# B&R Automation Studio project MotionTestBenchMaster (part 41)

```iecst
(* Input Signals *)
xInputAuto					:= stFillerModule.iq_stCmd.i_xAutoMode;
xInputJogMulti				:= stFillerModule.iq_stCmd.i_xJogMultiMode;
xInputAutoMulti				:= stFillerModule.iq_stCmd.i_xAutoMultiMode;
xInputSelHoming				:= stFillerModule.iq_stCmd.i_xSelectiveHomingMode;
xInputVelocity				:= stFillerModule.iq_stCmd.i_xVelocityMode;
xInputPositioning			:= stFillerModule.iq_stCmd.i_xPositioningMode;
xInputThirdPartySetup		:= stFillerModule.iq_stCmd.i_xThirdPartySetup;
xInputInductionSetup		:= stFillerModule.iq_stCmd.i_xInductionSetup;
xInputSlowMotion			:= stFillerModule.iq_stCmd.i_xSlowMotionForward OR stFillerModule.iq_stCmd.i_xSlowMotionBackward;
xInputBrakeRelease			:= stFillerModule.iq_stCmd.i_xBrakeRelease;
xInputStepByStep			:= stFillerModule.iq_stCmd.i_xStepByStep;
xInputStepByStepSingleAxis	:= stFillerModule.iq_stCmd.i_xStepByStepSingleAxis;//V4.A.A.1.7.0 Footbar
END_STEP
STEP ModeSelection:
(* Operating modes bits *)
xNoOpActive				:= TRUE;
xAutoActive 			:= FALSE;
xPositioningActive 		:= FALSE;
xSelHomingActive 		:= FALSE;
xBrakeReleaseActive 	:= FALSE;
xSlowMotionActive 		:= FALSE;
xJogMultiActive 		:= FALSE;
xAutoMultiActive 		:= FALSE;
xStepByStepActive 		:= FALSE;
xThirdPartySetupActive	:= FALSE;
xInductionSetupActive	:= FALSE;

(* Change status *)
xModeReady	:= usiMasterRequest = usiMasterStatus	AND
				NOT xAutoMode 						AND
				NOT xPositioningMode 				AND
				NOT xSelectiveHomingMode			AND
				NOT xVelocityMode					AND
				NOT xPositioningMode				AND
				NOT xStepByStepMode					AND
				NOT xJogMultiMode					AND
				NOT xAutoMultiMode					AND
				NOT xSlowMotionMode					AND
				NOT xThirdPartySetupMode			AND
				NOT xInductionSetupMode				AND
				NOT tofReactionActive.Q;

IF xModeReady THEN
	(* Local Master Request *)
	IF xInputJogMulti OR xInputAutoMulti THEN
		usiMasterRequest	:= LOCAL_MASTER;
	ELSIF xInputAuto OR	xInputPositioning OR xInputSelHoming OR xInputStepByStep OR xInputVelocity OR xInputThirdPartySetup OR xInputInductionSetup THEN
		usiMasterRequest	:= GLOBAL_MASTER;
	END_IF

	IF usiMasterStatus = GLOBAL_MASTER THEN
		IF xInputAuto THEN
			xAutoMode				:= TRUE;
		ELSIF xInputPositioning THEN
			xPositioningMode		:= TRUE;
		ELSIF xInputSelHoming THEN
			xSelectiveHomingMode	:= TRUE;
		ELSIF xInputThirdPartySetup THEN
			xThirdPartySetupMode	:= TRUE;
		ELSIF xInputInductionSetup THEN
			xInductionSetupMode		:= TRUE;
		ELSIF xInputStepByStep THEN
			xStepByStepMode			:= TRUE;
		ELSIF xInputVelocity THEN
			xVelocityMode			:= TRUE;
		END_IF
	ELSIF usiMasterStatus = LOCAL_MASTER THEN
		IF xInputJogMulti THEN
			xJogMultiMode 			:= TRUE;
		ELSIF xInputAutoMulti THEN
			xAutoMultiMode 			:= TRUE;
		ELSIF xInputSlowMotion THEN
			xSlowMotionMode			:= TRUE;
		END_IF
	END_IF
ELSIF tofReactionActive.Q THEN
	xBrakeReleaseMode	:= xInputBrakeRelease;
END_IF
END_STEP
ENTRY_ACTION
xExitStep	:= FALSE;
uiAutoStep	:= 0;
stFillerModule.iq_stStatus.q_xMasterRephased := FALSE;
END_ACTION
EXIT_ACTION
xNoOpActive	:= FALSE;
END_ACTION
TRANSITION FROM ModeSelection TO Auto:=
xAutoMode
END_TRANSITION
TRANSITION FROM ModeSelection TO Positioning:=
xPositioningMode
END_TRANSITION
STEP Positioning:
IF xReactionActive OR NOT xInputPositioning THEN
	xPositioningMode	:= FALSE;
END_IF

xPositioningActive	:= TRUE;

CASE uiPositioningStep OF
	0:
		IF stFillerModule.iq_stStatus.q_xRealAxesReadyForACommand AND stFillerModule.iq_astSubModuleAxis[CST_ModuleMasterAxis].iq_stStatus.q_stMainAxisStatus.q_xReadyForACommand THEN
			IF NOT stFillerModule.iq_stStatus.q_xSynchroWithOffset THEN
				uiPositioningStep	:= 100;
			ELSE
				uiPositioningStep	:= 50;
			END_IF
		END_IF

	50:
		FOR uiAxisIndex	:= uiFirstFillerModuleAxis TO uiLastFillerModuleAxis BY 1 DO
			stFillerModule.iq_astSubModuleAxis[uiAxisIndex].iq_stCmd.i_xPhaseCompensation := stFillerModule.iq_astSubModuleAxis[uiAxisIndex].iq_stStatus.q_stMainAxisStatus.q_xSynchroWithOffset;
		END_FOR

		IF NOT stFillerModule.iq_stStatus.q_xSynchroWithOffset THEN
			uiPositioningStep := 60;
		END_IF

	60:
		FOR uiAxisIndex	:= uiFirstFillerModuleAxis TO uiLastFillerModuleAxis BY 1 DO
			stFillerModule.iq_astSubModuleAxis[uiAxisIndex].iq_stCmd.i_xPhaseCompensation := FALSE;
		END_FOR
		uiPositioningStep := 100;

	100:
		IF stFillerModule.iq_stParameters.i_uiAxisSelected >= uiFirstFillerModuleAxis AND stFillerModule.iq_stParameters.i_uiAxisSelected <= uiLastFillerModuleAxis THEN
			uiOldAxisSelected := stFillerModule.iq_stParameters.i_uiAxisSelected;
			IF stFillerModule.iq_astSubModuleAxis[uiOldAxisSelected].iq_stStatus.q_stMainAxisStatus.q_xAxisReal THEN
				uiPositioningStep := 110;
			END_IF
		END_IF

	110:
		IF stFillerModule.iq_stCmd.i_xStepByStepSingleAxis THEN //V4.A.A.1.7.0 Footbar
			stFillerModule.iq_astSubModuleAxis[uiOldAxisSelected].iq_stParam.i_rPositioningVelocity	:= 10 * CST_PositioningVel ;
			stFillerModule.iq_astSubModuleAxis[uiOldAxisSelected].iq_stParam.i_rPositioningAccDec	:= 3 * CST_PositioningAccDec;
			stFillerModule.iq_astSubModuleAxis[uiOldAxisSelected].iq_stParam.i_lrAdditiveDistance	:= stFillerModule.iq_stParameters.i_rPositioningOffset;
		ELSE
			stFillerModule.iq_astSubModuleAxis[uiOldAxisSelected].iq_stParam.i_rPositioningVelocity	:= CST_PositioningVel;
			stFillerModule.iq_astSubModuleAxis[uiOldAxisSelected].iq_stParam.i_rPositioningAccDec	:= CST_PositioningAccDec;
			stFillerModule.iq_astSubModuleAxis[uiOldAxisSelected].iq_stParam.i_lrAdditiveDistance	:= stFillerModule.iq_stParameters.i_rPositioningOffset;
		END_IF

		IF stFillerModule.iq_astSubModuleAxis[uiOldAxisSelected].iq_stParam.i_lrAdditiveDistance = 0 THEN
			stFillerModule.iq_astSubModuleAxis[uiOldAxisSelected].iq_stParam.i_lrAdditiveDistance := 360.0;
		END_IF

		stFillerModule.iq_astSubModuleAxis[uiOldAxisSelected].iq_stCmd.i_xMoveAdditive	:= TRUE;

		tonPositDone(IN := FALSE, PT := T#5s);
		uiPositioningStep := 120;

	120:
		tonPositDone(IN := TRUE, PT := T#5s);
		IF NOT stFillerModule.iq_stStatus.q_xModuleStopped OR tonPositDone.Q THEN
			uiPositioningStep := 130;
		END_IF

	130:
		IF stFillerModule.iq_stStatus.q_xModuleStopped THEN
			stFillerModule.iq_astSubModuleAxis[uiOldAxisSelected].iq_stCmd.i_xMoveAdditive := FALSE;
			uiPositioningStep := 140;
		END_IF

	140:
		stFillerModule.iq_stStatus.q_xPositioningDone := TRUE;
END_CASE
END_STEP
ENTRY_ACTION
uiPositioningStep	:= 0;
END_ACTION
EXIT_ACTION
stFillerModule.iq_stStatus.q_xPositioningDone := FALSE;
stFillerModule.iq_astSubModuleAxis[uiOldAxisSelected].iq_stParam.i_rPositioningVelocity	:= CST_PositioningVel;//V4.A.A.1.7.0 Footbar
stFillerModule.iq_astSubModuleAxis[uiOldAxisSelected].iq_stParam.i_rPositioningAccDec	:= CST_PositioningAccDec;//V4.A.A.1.7.0 Footbar
END_ACTION
TRANSITION FROM Positioning TO PositExit:=
NOT xPositioningMode
END_TRANSITION
STEP PositExit:
stFillerModule.iq_astSubModuleAxis[uiOldAxisSelected].iq_stCmd.i_xMoveAdditive := FALSE;
stFillerModule.iq_stStatus.q_xPositioningDone := FALSE;
xExitStep := TRUE;
END_STEP
TRANSITION FROM PositExit TO ModeSelection:=
xExitStep
END_TRANSITION
(* @SFCISJUMP := 'ModeSelection' *)
TRANSITION FROM ModeSelection TO Velocity:=
xVelocityMode
END_TRANSITION
STEP Velocity:
IF xReactionActive OR NOT xInputVelocity THEN
	xVelocityMode	:= FALSE;
END_IF

xVelocityActive	:= TRUE;

CASE uiVelocityStep OF
	0:
		IF stFillerModule.iq_stStatus.q_xRealAxesReadyForACommand THEN
			uiVelocityStep	:= 100;
		END_IF

	100:
		IF stFillerModule.iq_stParameters.i_uiAxisSelected >= uiFirstFillerModuleAxis AND stFillerModule.iq_stParameters.i_uiAxisSelected <= uiLastFillerModuleAxis THEN
			uiOldAxisSelected	:= stFillerModule.iq_stParameters.i_uiAxisSelected;
			IF stFillerModule.iq_astSubModuleAxis[uiOldAxisSelected].iq_stStatus.q_stMainAxisStatus.q_xAxisReal THEN
				uiVelocityStep	:= 110;
			END_IF
		END_IF

	110:
		stFillerModule.iq_astSubModuleAxis[uiOldAxisSelected].iq_stParam.i_rEndlessVelocity		:= stFillerModule.iq_stParameters.i_rManualVelocity;

		stFillerModule.iq_astSubModuleAxis[uiOldAxisSelected].iq_stParam.i_lrAdditiveDistance	:= stFillerModule.iq_stParameters.i_rPositioningOffset;
		stFillerModule.iq_astSubModuleAxis[uiOldAxisSelected].iq_stCmd.i_xMoveVelocity			:= stFillerModule.iq_stCmd.i_xStart;
		uiVelocityStep	:= 120;

	120:
END_CASE
END_STEP
ENTRY_ACTION
uiVelocityStep	:= 0;
END_ACTION
EXIT_ACTION
xVelocityActive		:= FALSE;
uiOldAxisSelected	:= LIMIT(CST_FirstFillerModuleAxis, uiOldAxisSelected, CST_LastFillerModuleAxis);
stFillerModule.iq_astSubModuleAxis[uiOldAxisSelected].iq_stCmd.i_xMoveVelocity	:= FALSE;
END_ACTION
TRANSITION FROM Velocity TO VelExit:=
NOT xVelocityMode
END_TRANSITION
STEP VelExit:
xExitStep	:= stFillerModule.iq_stStatus.q_xModuleStopped;
END_STEP
TRANSITION FROM VelExit TO ModeSelection:=
xExitStep
END_TRANSITION
(* @SFCISJUMP := 'ModeSelection' *)
TRANSITION FROM ModeSelection TO SelHome:=
xSelectiveHomingMode
END_TRANSITION
STEP SelHome:
IF xReactionActive OR NOT xInputSelHoming THEN
	xSelectiveHomingMode := FALSE;
END_IF

xSelHomingActive	:= TRUE;

CASE uiSelectiveHomeStep OF
	0:
		IF stFillerModule.iq_stParameters.i_uiAxisSelected >= uiFirstFillerModuleAxis AND stFillerModule.iq_stParameters.i_uiAxisSelected <= uiLastFillerModuleAxis THEN
			uiOldAxisSelected	:= stFillerModule.iq_stParameters.i_uiAxisSelected;
			IF stFillerModule.iq_astSubModuleAxis[uiOldAxisSelected].iq_stStatus.q_stMainAxisStatus.q_xAxisReal THEN
				uiSelectiveHomeStep	:= 10;
			END_IF
		END_IF

	10:
		stFillerModule.iq_astSubModuleAxis[uiOldAxisSelected].iq_stCmd.i_xHome	:= TRUE;
		IF NOT stFillerModule.iq_astSubModuleAxis[uiOldAxisSelected].iq_stStatus.q_stMainAxisStatus.q_xIsHomed THEN
			uiSelectiveHomeStep	:= 20;
		END_IF

	20:
		uiSelectiveHomeStep	:= 30;

	30:
		IF stFillerModule.iq_astSubModuleAxis[uiOldAxisSelected].iq_stStatus.q_stMainAxisStatus.q_xIsHomed THEN
			stFillerModule.iq_astSubModuleAxis[uiOldAxisSelected].iq_stCmd.i_xHome	:= FALSE;
			uiSelectiveHomeStep	:= 40;
		END_IF

	40:
		stFillerModule.iq_stStatus.q_xSelHomingDone	:= TRUE;
END_CASE
END_STEP
ENTRY_ACTION
uiSelectiveHomeStep	:= 0;

(* Selective Homing done *)
stFillerModule.iq_stStatus.q_xSelHomingDone	:= FALSE;
END_ACTION
EXIT_ACTION
(* Selective Homing done *)
stFillerModule.iq_stStatus.q_xSelHomingDone	:= FALSE;
END_ACTION
TRANSITION FROM SelHome TO SelHomeExit:=
NOT xSelectiveHomingMode
END_TRANSITION
STEP SelHomeExit:
stFillerModule.iq_astSubModuleAxis[uiOldAxisSelected].iq_stCmd.i_xHome	:= FALSE;
xExitStep	:= TRUE;
END_STEP
TRANSITION FROM SelHomeExit TO ModeSelection:=
xExitStep
END_TRANSITION
(* @SFCISJUMP := 'ModeSelection' *)
TRANSITION FROM ModeSelection TO Brake:=
xBrakeReleaseMode
END_TRANSITION
STEP Brake:
xBrakeReleaseActive	:= TRUE;

IF NOT xInputBrakeRelease THEN
	xBrakeReleaseMode	:= FALSE;
END_IF

xBrakeReleaseActive	:= TRUE;

CASE uiBrakeReleaseStep OF
	0:
		uiOldAxisSelected	:= 0;
		IF stFillerModule.iq_stParameters.i_uiAxisSelected >= uiFirstFillerModuleAxis AND stFillerModule.iq_stParameters.i_uiAxisSelected <= uiLastFillerModuleAxis THEN
			uiOldAxisSelected	:= stFillerModule.iq_stParameters.i_uiAxisSelected;
			IF stFillerModule.iq_astSubModuleAxis[uiOldAxisSelected].iq_stStatus.q_stMainAxisStatus.q_xAxisReal THEN
				IF stFillerModule.iq_astSubModuleAxis[uiOldAxisSelected].iq_stStatus.q_stMainAxisStatus.q_xMotorWithBrake THEN
					uiBrakeReleaseStep	:= 100;
				ELSE
					uiBrakeReleaseStep	:= 400;
				END_IF
			END_IF
		END_IF

	100:
		stFillerModule.iq_astSubModuleAxis[uiOldAxisSelected].iq_stCmd.i_xReleaseBrake	:= TRUE;
		IF stFillerModule.iq_astSubModuleAxis[uiOldAxisSelected].iq_stStatus.q_stMainAxisStatus.q_xBrakeReleased THEN
			uiBrakeReleaseStep	:= 200;
		END_IF

	200:
		stFillerModule.iq_stStatus.q_xBrakeReleaseDone	:= TRUE;

	400:
		stFillerModule.iq_stStatus.q_xBrakeReleaseDone	:=	TRUE;
END_CASE
END_STEP
ENTRY_ACTION
uiBrakeReleaseStep	:= 0;
END_ACTION
EXIT_ACTION
xBrakeReleaseActive	:= FALSE;
stFillerModule.iq_stStatus.q_xBrakeReleaseDone	:= FALSE;

IF uiOldAxisSelected <> 0 THEN
	stFillerModule.iq_astSubModuleAxis[uiOldAxisSelected].iq_stCmd.i_xReleaseBrake	:= FALSE;
END_IF
END_ACTION
TRANSITION FROM Brake TO BrakeExit:=
NOT xBrakeReleaseMode
END_TRANSITION
STEP BrakeExit:
xExitStep	:= TRUE;
END_STEP
TRANSITION FROM BrakeExit TO ModeSelection:=
xExitStep
END_TRANSITION
(* @SFCISJUMP := 'ModeSelection' *)
TRANSITION FROM ModeSelection TO ThirdPartySetup:=
xThirdPartySetupMode
END_TRANSITION
STEP ThirdPartySetup:
IF xReactionActive OR NOT xInputThirdPartySetup THEN
	xThirdPartySetupMode	:= FALSE;
END_IF

xThirdPartySetupActive	:= TRUE;

CASE uiThirdPartySetupStep OF
	0:
		IF stFillerModule.iq_stParameters.i_uiAxisSelected >= uiFirstFillerModuleAxis AND stFillerModule.iq_stParameters.i_uiAxisSelected <= uiLastFillerModuleAxis THEN
			uiOldAxisSelected	:= stFillerModule.iq_stParameters.i_uiAxisSelected;
			IF stFillerModule.iq_astSubModuleAxis[uiOldAxisSelected].iq_stStatus.q_stMainAxisStatus.q_xAxisReal AND stFillerModule.iq_astSubModuleAxis[uiOldAxisSelected].iq_stStatus.q_stMainAxisStatus.q_xThirdPartyMotor THEN
				uiThirdPartySetupStep	:= 10;
			ELSE
				uiThirdPartySetupStep	:= 40;
			END_IF
		END_IF

	10:
		stFillerModule.iq_astSubModuleAxis[uiOldAxisSelected].iq_stCmd.i_xThirdPartySetup	:= TRUE;
		IF NOT stFillerModule.iq_astSubModuleAxis[uiOldAxisSelected].iq_stStatus.q_stMainAxisStatus.q_xMotorSetupDone THEN
			uiThirdPartySetupStep	:= 20;
		END_IF

	20:
		IF stFillerModule.iq_astSubModuleAxis[uiOldAxisSelected].iq_stStatus.q_stMainAxisStatus.q_xMotorSetupDone THEN
			stFillerModule.iq_astSubModuleAxis[uiOldAxisSelected].iq_stCmd.i_xThirdPartySetup	:= FALSE;
			uiThirdPartySetupStep	:= 40;
		END_IF

	40:
		stFillerModule.iq_stStatus.q_xThirdPartySetupDone := TRUE;
END_CASE
END_STEP
ENTRY_ACTION
uiThirdPartySetupStep	:= 0;
END_ACTION
EXIT_ACTION
stFillerModule.iq_stStatus.q_xThirdPartySetupDone := FALSE;
END_ACTION
TRANSITION FROM ThirdPartySetup TO ThirdPartySetupExit:=
NOT xThirdPartySetupMode
END_TRANSITION
STEP ThirdPartySetupExit:
stFillerModule.iq_astSubModuleAxis[uiOldAxisSelected].iq_stCmd.i_xThirdPartySetup	:= FALSE;
stFillerModule.iq_stStatus.q_xThirdPartySetupDone := FALSE;
stFillerModule.iq_stStatus.q_xThirdPartySetupActive := FALSE;
xExitStep := TRUE;
END_STEP
TRANSITION FROM ThirdPartySetupExit TO ModeSelection:=
xExitStep
END_TRANSITION
(* @SFCISJUMP := 'ModeSelection' *)
TRANSITION FROM ModeSelection TO InductionSetup:=
xInductionSetupMode
END_TRANSITION
STEP InductionSetup:
IF xReactionActive OR NOT xInputInductionSetup THEN
	xInductionSetupMode	:= FALSE;
END_IF

xInductionSetupActive	:= TRUE;

CASE uiInductionSetupStep OF
	0:
		IF stFillerModule.iq_stParameters.i_uiAxisSelected >= uiFirstFillerModuleAxis AND stFillerModule.iq_stParameters.i_uiAxisSelected <= uiLastFillerModuleAxis THEN
			uiOldAxisSelected	:= stFillerModule.iq_stParameters.i_uiAxisSelected;
			IF stFillerModule.iq_astSubModuleAxis[uiOldAxisSelected].iq_stStatus.q_stMainAxisStatus.q_xAxisReal AND stFillerModule.iq_astSubModuleAxis[uiOldAxisSelected].iq_stStatus.q_stMainAxisStatus.q_xInduction THEN
				uiInductionSetupStep	:= 10;
			ELSE
				uiInductionSetupStep	:= 40;
			END_IF
		END_IF

	10:
		stFillerModule.iq_astSubModuleAxis[uiOldAxisSelected].iq_stCmd.i_xInductionMotorSetup	:= TRUE;
		IF NOT stFillerModule.iq_astSubModuleAxis[uiOldAxisSelected].iq_stStatus.q_stMainAxisStatus.q_xMotorSetupDone THEN
			uiInductionSetupStep	:= 20;
		END_IF

	20:
		IF stFillerModule.iq_astSubModuleAxis[uiOldAxisSelected].iq_stStatus.q_stMainAxisStatus.q_xMotorSetupDone THEN
			stFillerModule.iq_astSubModuleAxis[uiOldAxisSelected].iq_stCmd.i_xInductionMotorSetup	:= FALSE;
			uiInductionSetupStep	:= 40;
		END_IF

	40:
		stFillerModule.iq_stStatus.q_xInductionSetupDone := TRUE;
END_CASE
END_STEP
ENTRY_ACTION
uiInductionSetupStep	:= 0;
END_ACTION
EXIT_ACTION
stFillerModule.iq_stStatus.q_xInductionSetupDone := FALSE;
END_ACTION
TRANSITION FROM InductionSetup TO InductionSetupExit1:=
NOT xInductionSetupMode
END_TRANSITION
STEP InductionSetupExit1:
stFillerModule.iq_astSubModuleAxis[uiOldAxisSelected].iq_stCmd.i_xInductionMotorSetup	:= FALSE;
stFillerModule.iq_stStatus.q_xInductionSetupDone := FALSE;
stFillerModule.iq_stStatus.q_xInductionSetupActive := FALSE;
xExitStep := TRUE;
END_STEP
TRANSITION FROM InductionSetupExit1 TO ModeSelection:=
xExitStep
END_TRANSITION
(* @SFCISJUMP := 'ModeSelection' *)
TRANSITION FROM ModeSelection TO SlowMotion:=
xSlowMotionMode
END_TRANSITION
STEP SlowMotion:
IF xReactionActive OR NOT (stFillerModule.iq_stCmd.i_xSlowMotionForward OR stFillerModule.iq_stCmd.i_xSlowMotionBackward) THEN
	xSlowMotionMode	:= FALSE;
END_IF

xSlowMotionActive	:= TRUE;

CASE uiSlowMotionStep OF
	0:
END_CASE
END_STEP
ENTRY_ACTION
uiSlowMotionStep	:= 0;
END_ACTION
EXIT_ACTION
stFillerModule.iq_astSubModuleAxis[CST_MainAxis].iq_stCmd.i_xSlowMotionFwd	:= FALSE;
stFillerModule.iq_astSubModuleAxis[CST_MainAxis].iq_stCmd.i_xSlowMotionBwd	:= FALSE;
xSlowMotionActive	:= FALSE;
END_ACTION
TRANSITION FROM SlowMotion TO SlowMotionExit:=
NOT xSlowMotionMode
END_TRANSITION
STEP SlowMotionExit:
stFillerModule.iq_astSubModuleAxis[CST_ModuleMasterAxis].iq_stCmd.i_xSlowMotionBwd	:= FALSE;
stFillerModule.iq_astSubModuleAxis[CST_ModuleMasterAxis].iq_stCmd.i_xSlowMotionFwd	:= FALSE;

IF stFillerModule.iq_stStatus.q_xModuleStopped THEN
	FOR uiAxisIndex	:= CST_ModuleMasterAxis TO CST_LastFillerModuleAxis BY 1 DO
		stFillerModule.iq_astSubModuleAxis[uiAxisIndex].iq_stCmd.i_xGear 				:= FALSE;
		stFillerModule.iq_astSubModuleAxis[uiAxisIndex].iq_stCmd.i_xPhaseCompensation	:= FALSE;
	END_FOR
	xExitStep := NOT stFillerModule.iq_stStatus.q_xModuleSynchronized;
END_IF
END_STEP
TRANSITION FROM SlowMotionExit TO ModeSelection:=
xExitStep
END_TRANSITION
(* @SFCISJUMP := 'ModeSelection' *)
TRANSITION FROM ModeSelection TO JogMulti:=
xJogMultiMode
END_TRANSITION
STEP JogMulti:
IF xReactionActive OR NOT xInputJogMulti THEN
	xJogMultiMode	:= FALSE;
END_IF

xJogMultiActive	:= TRUE;

CASE uiJogMulti OF
	0:
		IF stFillerModule.iq_stStatus.q_xRealAxesReadyForACommand AND stFillerModule.iq_astSubModuleAxis[CST_ModuleMasterAxis].iq_stStatus.q_stMainAxisStatus.q_xReadyForACommand THEN
			IF NOT stFillerModule.iq_stStatus.q_xSynchroWithOffset THEN
				uiJogMulti	:= 100;
			ELSE
				uiJogMulti	:= 50;
			END_IF
		END_IF

	50:
		FOR uiAxisIndex	:= uiFirstFillerModuleAxis	TO uiLastFillerModuleAxis BY 1 DO
			stFillerModule.iq_astSubModuleAxis[uiAxisIndex].iq_stCmd.i_xPhaseCompensation := stFillerModule.iq_astSubModuleAxis[uiAxisIndex].iq_stStatus.q_stMainAxisStatus.q_xSynchroWithOffset;
		END_FOR
		uiJogMulti	:= 60;

	60:
		IF NOT stFillerModule.iq_stStatus.q_xSynchroWithOffset THEN
			uiJogMulti	:= 70;
		END_IF

	70:
		FOR uiAxisIndex	:= uiFirstFillerModuleAxis	TO uiLastFillerModuleAxis BY 1 DO
			stFillerModule.iq_astSubModuleAxis[uiAxisIndex].iq_stCmd.i_xPhaseCompensation := FALSE;
		END_FOR
		uiJogMulti	:= 100;

	100:
		IF NOT stFillerModule.iq_stCmd.i_xStart THEN
			IF stFillerModule.iq_stCmd.i_xMasterRephasingRequest THEN
				stFillerModule.iq_astSubModuleAxis[CST_ModuleMasterAxis].iq_stCmd.i_xHome	:= TRUE;
				uiJogMulti	:= 105;
			END_IF
		END_IF

	105:
		IF NOT stFillerModule.iq_astSubModuleAxis[CST_ModuleMasterAxis].iq_stStatus.q_stMainAxisStatus.q_xIsHomed THEN
			uiJogMulti	:= 110;
		END_IF

	110:
		IF stFillerModule.iq_astSubModuleAxis[CST_ModuleMasterAxis].iq_stStatus.q_stMainAxisStatus.q_xIsHomed THEN
			stFillerModule.iq_stStatus.q_xMasterRephased								:= TRUE;
			stFillerModule.iq_astSubModuleAxis[CST_ModuleMasterAxis].iq_stCmd.i_xHome	:= FALSE;
			uiJogMulti	:= 120;
		END_IF

	120:
		IF stFillerModule.iq_stCmd.i_xJogPB THEN
			FOR uiAxisIndex	:= uiFirstFillerModuleAxis TO uiLastFillerModuleAxis BY 1 DO
				stFillerModule.iq_astSubModuleAxis[uiAxisIndex].iq_stCmd.i_xGear := stFillerModule.iq_astSubModuleAxis[uiAxisIndex].iq_stStatus.q_stMainAxisStatus.q_xAxisReal;
			END_FOR
			uiJogMulti	:= 130;
		END_IF

	130:
		(* Wait for real axes synchronized *)
		IF stFillerModule.iq_stStatus.q_xRealAxesSynchronized THEN
			uiJogMulti	:= 140;
		END_IF

	140:(* Step JOG MULTI *)
		stFillerModule.iq_astSubModuleAxis[CST_ModuleMasterAxis].iq_stParam.i_rJogVelocity	:= MAX(1, stFillerModule.iq_stParameters.i_rJogVelocity);
		stFillerModule.iq_astSubModuleAxis[CST_ModuleMasterAxis].iq_stCmd.i_xJogPositive	:= stFillerModule.iq_stCmd.i_xJogPB;

		IF NOT stFillerModule.iq_stCmd.i_xJogPB THEN
			uiJogMulti	:= 150;
		END_IF

	150:
END_CASE
END_STEP
ENTRY_ACTION
uiJogMulti	:= 0;
END_ACTION
EXIT_ACTION
stFillerModule.iq_stStatus.q_xMasterRephased										:= FALSE;
stFillerModule.iq_astSubModuleAxis[CST_ModuleMasterAxis].iq_stCmd.i_xJogPositive	:= FALSE;
stFillerModule.iq_astSubModuleAxis[CST_ModuleMasterAxis].iq_stCmd.i_xHome			:= FALSE;
END_ACTION
TRANSITION FROM JogMulti TO JogExit:=
NOT xJogMultiMode
END_TRANSITION
STEP JogExit:
(* All axis commands are set to FALSE *)
stFillerModule.iq_astSubModuleAxis[CST_ModuleMasterAxis].iq_stCmd.i_xMoveVelocity	:= FALSE;
stFillerModule.iq_astSubModuleAxis[CST_ModuleMasterAxis].iq_stCmd.i_xJogPositive	:= FALSE;
stFillerModule.iq_astSubModuleAxis[CST_ModuleMasterAxis].iq_stCmd.i_xQuickStop		:= TRUE;
stFillerModule.iq_astSubModuleAxis[CST_ModuleMasterAxis].iq_stCmd.i_xHome			:= FALSE;

(* Axis Stopped all real axis are set in GearOut mode *)
IF stFillerModule.iq_stStatus.q_xModuleStopped THEN
	stFillerModule.iq_astSubModuleAxis[CST_ModuleMasterAxis].iq_stCmd.i_xQuickStop	:= FALSE;
	FOR uiAxisIndex	:= CST_FirstFillerModuleAxis TO CST_LastFillerModuleAxis BY 1 DO
		stFillerModule.iq_astSubModuleAxis[uiAxisIndex].iq_stCmd.i_xGear 				:= FALSE;
		stFillerModule.iq_astSubModuleAxis[uiAxisIndex].iq_stCmd.i_xPhaseCompensation	:= FALSE;
	END_FOR
	xExitStep	:= NOT stFillerModule.iq_stStatus.q_xRealAxesSynchronized;
END_IF
END_STEP
TRANSITION FROM JogExit TO ModeSelection:=
xExitStep
END_TRANSITION
(* @SFCISJUMP := 'ModeSelection' *)
TRANSITION FROM ModeSelection TO AutoMulti:=
xAutoMultiMode
END_TRANSITION
STEP AutoMulti:
IF xReactionActive OR NOT xInputAutoMulti THEN
	xAutoMultiMode	:= FALSE;
END_IF

xAutoMultiActive	:= TRUE;

CASE uiAutoMulti OF
	0:
		IF stFillerModule.iq_stStatus.q_xRealAxesReadyForACommand AND stFillerModule.iq_astSubModuleAxis[CST_ModuleMasterAxis].iq_stStatus.q_stMainAxisStatus.q_xReadyForACommand THEN
			IF NOT stFillerModule.iq_stStatus.q_xSynchroWithOffset THEN
				uiAutoMulti	:= 100;
			ELSE
				uiAutoMulti	:= 50;
			END_IF
		END_IF

	50:
		FOR uiAxisIndex	:= uiFirstFillerModuleAxis TO uiLastFillerModuleAxis BY 1 DO
			stFillerModule.iq_astSubModuleAxis[uiAxisIndex].iq_stCmd.i_xPhaseCompensation := stFillerModule.iq_astSubModuleAxis[uiAxisIndex].iq_stStatus.q_stMainAxisStatus.q_xSynchroWithOffset;
		END_FOR
		uiAutoMulti	:= 60;

	60:
		IF NOT stFillerModule.iq_stStatus.q_xSynchroWithOffset THEN
			uiAutoMulti	:= 70;
		END_IF

	70:
		FOR uiAxisIndex	:= uiFirstFillerModuleAxis TO uiLastFillerModuleAxis BY 1 DO
			stFillerModule.iq_astSubModuleAxis[uiAxisIndex].iq_stCmd.i_xPhaseCompensation := FALSE;
		END_FOR
		uiAutoMulti	:= 100;

	100:
		IF stFillerModule.iq_stCmd.i_xMasterRephasingRequest THEN
			uiAutoMulti	:= 105;
		END_IF

	105:
		stFillerModule.iq_astSubModuleAxis[CST_ModuleMasterAxis].iq_stCmd.i_xHome := TRUE;
		uiAutoMulti	:= 110;

	110:
		stFillerModule.iq_stStatus.q_xMasterRephased := TRUE;
		uiAutoMulti	:= 115;

	115:
		IF stFillerModule.iq_astSubModuleAxis[CST_ModuleMasterAxis].iq_stStatus.q_stMainAxisStatus.q_xIsHomed THEN
			stFillerModule.iq_astSubModuleAxis[CST_ModuleMasterAxis].iq_stCmd.i_xHome := FALSE;
			uiAutoMulti	:= 120;
		END_IF

	120:
		IF stFillerModule.iq_stCmd.i_xStart THEN
			FOR uiAxisIndex	:= uiFirstFillerModuleAxis TO uiLastFillerModuleAxis BY 1 DO
				IF NOT stFillerModule.iq_astSubModuleAxis[uiAxisIndex].iq_stStatus.q_stMainAxisStatus.q_xVelocityControl THEN
					stFillerModule.iq_astSubModuleAxis[uiAxisIndex].iq_stCmd.i_xGear := stFillerModule.iq_astSubModuleAxis[uiAxisIndex].iq_stStatus.q_stMainAxisStatus.q_xAxisReal;
				ELSE
					stFillerModule.iq_astSubModuleAxis[uiAxisIndex].iq_stCmd.i_xGear := NOT stFillerModule.iq_stCmd.i_xVelocityAxisStop;
				END_IF
			END_FOR
		END_IF

		(* Wait for real axes synchronized *)
		IF stFillerModule.iq_stStatus.q_xRealAxesSynchronized THEN
			uiAutoMulti	:= 130;
		END_IF

	130:
		IF stFillerModule.iq_stStatus.q_xSynchroWithOffset AND stFillerModule.iq_stCmd.i_xPhaseCompensation THEN
			uiAutoMulti	:= 300;
		ELSIF stFillerModule.iq_stCmd.i_xStart THEN
			uiAutoMulti	:= 140;
		END_IF

	140:(* Step AUTO MULTI *)
		stFillerModule.iq_astSubModuleAxis[CST_ModuleMasterAxis].iq_stParam.i_rEndlessVelocity	:= MAX(1, stFillerModule.iq_stParameters.i_rEndlessVelocity);
		stFillerModule.iq_astSubModuleAxis[CST_ModuleMasterAxis].iq_stCmd.i_xMoveVelocity		:= stFillerModule.iq_stCmd.i_xStart;

		IF NOT stFillerModule.iq_stCmd.i_xStart THEN
			uiAutoMulti	:= 150;
		ELSIF NOT stFillerModule.iq_stStatus.q_xModuleStopped THEN
			uiOldAxisSelected := LIMIT(uiFirstFillerModuleAxis, stFillerModule.iq_stParameters.i_uiAxisSelected, uiLastFillerModuleAxis);
			IF stFillerModule.iq_stParameters.i_uiAxisSelected >=  uiFirstFillerModuleAxis 	AND
				stFillerModule.iq_stParameters.i_uiAxisSelected <=	uiLastFillerModuleAxis 	AND
				stFillerModule.iq_astSubModuleAxis[uiOldAxisSelected].iq_stStatus.q_stMainAxisStatus.q_xAxisReal THEN
				IF stFillerModule.iq_stCmd.i_xOnePitchShift THEN
					stFillerModule.iq_astSubModuleAxis[uiOldAxisSelected].iq_stCmd.i_xOnePitchShift := TRUE;
					uiAutoMulti	:= 160;
				ELSIF stFillerModule.iq_stCmd.i_xPhaseShift AND stFillerModule.iq_stParameters.i_rPhaseShiftDistance <> 0 THEN
					stFillerModule.iq_astSubModuleAxis[uiOldAxisSelected].iq_stParam.i_rPhaseShiftDistance 	:= stFillerModule.iq_stParameters.i_rPhaseShiftDistance;
					stFillerModule.iq_astSubModuleAxis[uiOldAxisSelected].iq_stCmd.i_xPhaseShift			:= TRUE;
					uiAutoMulti	:= 180;
				END_IF
			END_IF
		END_IF

	150:
		IF stFillerModule.iq_stStatus.q_xModuleStopped THEN
			uiAutoMulti	:= 130;
		END_IF

	160:(* One pitch shift *)
		IF NOT stFillerModule.iq_astSubModuleAxis[uiOldAxisSelected].iq_stStatus.q_stMainAxisStatus.q_xPhaseShiftDone AND NOT stFillerModule.iq_stCmd.i_xOnePitchShift THEN
			stFillerModule.iq_astSubModuleAxis[uiOldAxisSelected].iq_stCmd.i_xOnePitchShift := FALSE;
			uiAutoMulti	:= 140;
		END_IF

	180:(* Phase shift *)
		IF stFillerModule.iq_astSubModuleAxis[uiOldAxisSelected].iq_stStatus.q_stMainAxisStatus.q_xPhaseShiftDone AND NOT stFillerModule.iq_stCmd.i_xPhaseShift THEN
			stFillerModule.iq_astSubModuleAxis[uiOldAxisSelected].iq_stCmd.i_xPhaseShift 	:= FALSE;
			uiAutoMulti	:= 140;
		END_IF

	300:(* Phase Offset Compensations *)
		FOR uiAxisIndex	:= uiFirstFillerModuleAxis TO uiLastFillerModuleAxis BY 1 DO
			IF stFillerModule.iq_astSubModuleAxis[uiAxisIndex].iq_stStatus.q_stMainAxisStatus.q_xSynchroWithOffset THEN
				stFillerModule.iq_astSubModuleAxis[uiAxisIndex].iq_stCmd.i_xGear 				:= FALSE;
				stFillerModule.iq_astSubModuleAxis[uiAxisIndex].iq_stCmd.i_xPhaseCompensation	:= TRUE;
			END_IF
		END_FOR
		uiAutoMulti	:= 310;

	310:
		IF NOT stFillerModule.iq_stStatus.q_xSynchroWithOffset THEN
			FOR uiAxisIndex	:= uiFirstFillerModuleAxis TO uiLastFillerModuleAxis BY 1 DO
				IF NOT stFillerModule.iq_astSubModuleAxis[uiAxisIndex].iq_stStatus.q_stMainAxisStatus.q_xVelocityControl THEN
					stFillerModule.iq_astSubModuleAxis[uiAxisIndex].iq_stCmd.i_xGear := stFillerModule.iq_astSubModuleAxis[uiAxisIndex].iq_stStatus.q_stMainAxisStatus.q_xAxisReal;
				ELSE
					stFillerModule.iq_astSubModuleAxis[uiAxisIndex].iq_stCmd.i_xGear := NOT stFillerModule.iq_stCmd.i_xVelocityAxisStop;
				END_IF
				stFillerModule.iq_astSubModuleAxis[uiAxisIndex].iq_stCmd.i_xPhaseCompensation	:= FALSE;
			END_FOR
			uiAutoMulti := 130;
		END_IF
END_CASE

IF uiAutoStep > 120 AND EDGE(stFillerModule.iq_stCmd.i_xVelocityAxisStop) THEN
	FOR uiAxisIndex	:= uiFirstFillerModuleAxis TO uiLastFillerModuleAxis BY 1 DO
		IF stFillerModule.iq_astSubModuleAxis[uiAxisIndex].iq_stStatus.q_stMainAxisStatus.q_xVelocityControl THEN
			stFillerModule.iq_astSubModuleAxis[uiAxisIndex].iq_stCmd.i_xGear := NOT stFillerModule.iq_stCmd.i_xVelocityAxisStop;
		END_IF
	END_FOR
END_IF
END_STEP
ENTRY_ACTION
uiAutoMulti	:= 0;
END_ACTION
TRANSITION FROM AutoMulti TO AutoMultiExit:=
NOT xAutoMultiMode
END_TRANSITION
STEP AutoMultiExit:
(* All axis commands are set to FALSE *)
stFillerModule.iq_astSubModuleAxis[CST_ModuleMasterAxis].iq_stCmd.i_xMoveVelocity	:= FALSE;
stFillerModule.iq_astSubModuleAxis[CST_ModuleMasterAxis].iq_stCmd.i_xJogPositive	:= FALSE;
stFillerModule.iq_astSubModuleAxis[CST_ModuleMasterAxis].iq_stCmd.i_xHome			:= FALSE;

(* Axis Stopped all real axis are set in GearOut mode *)
IF stFillerModule.iq_stStatus.q_xModuleStopped THEN
	FOR uiAxisIndex	:= CST_FirstFillerModuleAxis TO uiLastFillerModuleAxis BY 1 DO
		stFillerModule.iq_astSubModuleAxis[uiAxisIndex].iq_stCmd.i_xGear 				:= FALSE;
		stFillerModule.iq_astSubModuleAxis[uiAxisIndex].iq_stCmd.i_xPhaseCompensation	:= FALSE;
	END_FOR
	xExitStep	:= NOT stFillerModule.iq_stStatus.q_xRealAxesSynchronized;
END_IF
END_STEP
TRANSITION FROM AutoMultiExit TO ModeSelection:=
xExitStep
END_TRANSITION
(* @SFCISJUMP := 'ModeSelection' *)
TRANSITION FROM ModeSelection TO StepByStep:=
xStepByStepMode
END_TRANSITION
STEP StepByStep:
IF xReactionActive OR NOT xInputStepByStep THEN
	xStepByStepMode	:= FALSE;
END_IF

xStepByStepActive	:= TRUE;

CASE uiStepByStep OF
	0:
		IF stFillerModule.iq_stCmd.i_xStart THEN
			uiStepByStep	:= 20;
		END_IF

	20:
		IF stFillerModule.iq_stStatus.q_xRealAxesReadyForACommand AND stFillerModule.iq_astSubModuleAxis[CST_ModuleMasterAxis].iq_stStatus.q_stMainAxisStatus.q_xReadyForACommand THEN
			IF NOT stFillerModule.iq_stStatus.q_xSynchroWithOffset THEN
				uiStepByStep	:= 100;
			ELSE
				uiStepByStep	:= 50;
			END_IF
		END_IF

	50:
		FOR uiAxisIndex	:= uiFirstFillerModuleAxis TO uiLastFillerModuleAxis BY 1 DO
			stFillerModule.iq_astSubModuleAxis[uiAxisIndex].iq_stCmd.i_xPhaseCompensation := stFillerModule.iq_astSubModuleAxis[CST_ModuleMasterAxis].iq_stStatus.q_stMainAxisStatus.q_xSynchroWithOffset;
		END_FOR

		IF NOT stFillerModule.iq_stStatus.q_xSynchroWithOffset THEN
			uiStepByStep	:= 60;
		END_IF

	60:
		FOR uiAxisIndex	:= uiFirstFillerModuleAxis TO uiLastFillerModuleAxis BY 1 DO
			stFillerModule.iq_astSubModuleAxis[uiAxisIndex].iq_stCmd.i_xPhaseCompensation := FALSE;
		END_FOR

		uiStepByStep	:= 100;

	100:
		FOR uiAxisIndex	:= uiFirstFillerModuleAxis TO uiLastFillerModuleAxis BY 1 DO
			stFillerModule.iq_astSubModuleAxis[uiAxisIndex].iq_stCmd.i_xGear := stFillerModule.iq_astSubModuleAxis[CST_ModuleMasterAxis].iq_stStatus.q_stMainAxisStatus.q_xAxisReal;
		END_FOR

		IF stFillerModule.iq_stStatus.q_xModuleSynchronized THEN
			uiStepByStep	:= 110;
		END_IF

	110:
		uiNumberOfSteps	:= MAX(1, stFillerModule.iq_stParameters.i_uiNumberOfSteps);
		rAxisDistance	:= LREAL_TO_REAL(stFillerModule.iq_stParameters.i_rStopPosition	- stFillerModule.iq_astSubModuleAxis[CST_ModuleMasterAxis].iq_stStatus.q_stMainAxisStatus.q_lrPosition);

		IF rAxisDistance < 0.0 THEN
			rAxisDistance	:= rAxisDistance + 360.0;
		END_IF

		IF rAxisDistance < 10.0 THEN
			rAxisDistance	:= 360.0 + rAxisDistance;
		END_IF

		uiStepByStep	:= 120;

	120:
		IF stFillerModule.iq_stCmd.i_xStart THEN
			stFillerModule.iq_astSubModuleAxis[CST_ModuleMasterAxis].iq_stParam.i_rPositioningVelocity	:= CST_PositioningVel;
			stFillerModule.iq_astSubModuleAxis[CST_ModuleMasterAxis].iq_stParam.i_rPositioningAccDec	:= CST_PositioningAccDec;
			stFillerModule.iq_astSubModuleAxis[CST_ModuleMasterAxis].iq_stCmd.i_xMoveAdditive			:= TRUE;
			uiStepByStep	:= 130;
		END_IF

	130:
		IF NOT stFillerModule.iq_stStatus.q_xModuleStopped THEN
			stFillerModule.iq_astSubModuleAxis[CST_ModuleMasterAxis].iq_stCmd.i_xMoveAdditive := FALSE;
			uiStepByStep	:= 140;
		END_IF

	140:
		IF stFillerModule.iq_stStatus.q_xModuleStopped AND stFillerModule.iq_stCmd.i_xStart THEN
			uiStepByStep	:= 110;
		END_IF
END_CASE

END_STEP
ENTRY_ACTION
uiStepByStep	:= 0;
END_ACTION
TRANSITION FROM StepByStep TO StepByStepExit:=
NOT xStepByStepMode
END_TRANSITION
STEP StepByStepExit:
stFillerModule.iq_astSubModuleAxis[CST_ModuleMasterAxis].iq_stCmd.i_xMoveAdditive	:= FALSE;
IF stFillerModule.iq_stStatus.q_xModuleStopped THEN
	FOR uiAxisIndex	:= uiFirstFillerModuleAxis TO uiLastFillerModuleAxis BY 1 DO
		stFillerModule.iq_astSubModuleAxis[uiAxisIndex].iq_stCmd.i_xGear 				:= FALSE;
		stFillerModule.iq_astSubModuleAxis[uiAxisIndex].iq_stCmd.i_xPhaseCompensation	:= FALSE;
	END_FOR
	xExitStep	:= NOT stFillerModule.iq_stStatus.q_xModuleSynchronized;
END_IF
END_STEP
TRANSITION FROM StepByStepExit TO ModeSelection:=
xExitStep
END_TRANSITION
(* @SFCISJUMP := 'ModeSelection' *)
STEP Auto:
IF xReactionActive OR NOT xInputAuto THEN
	xAutoMode	:= FALSE;
END_IF

xAutoActive	:= TRUE;

CASE uiAutoStep OF
	0:
		IF stFillerModule.iq_stStatus.q_xRealAxesReadyForACommand AND stFillerModule.iq_astSubModuleAxis[CST_ModuleMasterAxis].iq_stStatus.q_stMainAxisStatus.q_xReadyForACommand THEN
			IF NOT stFillerModule.iq_stStatus.q_xSynchroWithOffset THEN
				uiAutoStep	:= 100;
			ELSE
				uiAutoStep	:= 50;
			END_IF
		END_IF

	50:
		FOR uiAxisIndex	:= uiFirstFillerModuleAxis	TO uiLastFillerModuleAxis BY 1 DO
			stFillerModule.iq_astSubModuleAxis[uiAxisIndex].iq_stCmd.i_xPhaseCompensation := stFillerModule.iq_astSubModuleAxis[uiAxisIndex].iq_stStatus.q_stMainAxisStatus.q_xSynchroWithOffset;
		END_FOR
		uiAutoStep	:= 60;

	60:
		IF NOT stFillerModule.iq_stStatus.q_xSynchroWithOffset THEN
			uiAutoStep	:= 70;
		END_IF

	70:
		FOR uiAxisIndex	:= uiFirstFillerModuleAxis	TO uiLastFillerModuleAxis  BY 1 DO
			stFillerModule.iq_astSubModuleAxis[uiAxisIndex].iq_stCmd.i_xPhaseCompensation := FALSE;
		END_FOR
		uiAutoStep	:= 0;

	100:
		IF stFillerModule.iq_stCmd.i_xStart THEN
 			stFillerModule.iq_astSubModuleAxis[CST_ModuleMasterAxis].iq_stCmd.i_xHome 	:= TRUE;
			IF NOT stFillerModule.iq_astSubModuleAxis[CST_ModuleMasterAxis].iq_stStatus.q_stMainAxisStatus.q_xIsHomed THEN
				stFillerModule.iq_stStatus.q_xMasterRephased := TRUE;
				uiAutoStep	:= 110;
			END_IF
		END_IF

	110:
		IF stFillerModule.iq_astSubModuleAxis[CST_ModuleMasterAxis].iq_stStatus.q_stMainAxisStatus.q_xIsHomed THEN
			stFillerModule.iq_astSubModuleAxis[CST_ModuleMasterAxis].iq_stCmd.i_xHome 	:= FALSE;
			uiAutoStep	:= 120;
		END_IF

	120:
		FOR uiAxisIndex	:= uiFirstFillerModuleAxis TO uiLastFillerModuleAxis BY 1 DO
			IF NOT stFillerModule.iq_astSubModuleAxis[uiAxisIndex].iq_stStatus.q_stMainAxisStatus.q_xVelocityControl THEN
				stFillerModule.iq_astSubModuleAxis[uiAxisIndex].iq_stCmd.i_xGear := stFillerModule.iq_astSubModuleAxis[uiAxisIndex].iq_stStatus.q_stMainAxisStatus.q_xAxisReal;
			ELSE
				stFillerModule.iq_astSubModuleAxis[uiAxisIndex].iq_stCmd.i_xGear := NOT stFillerModule.iq_stCmd.i_xVelocityAxisStop;
			END_IF
		END_FOR

		IF stFillerModule.iq_stStatus.q_xRealAxesSynchronized THEN
			uiAutoStep	:= 130;
		END_IF

	130:(* If the machine is running the phasing command is taken in account *)
		IF NOT stFillerModule.iq_stStatus.q_xModuleStopped THEN
			uiOldAxisSelected	:= LIMIT(uiFirstFillerModuleAxis, stFillerModule.iq_stParameters.i_uiAxisSelected, uiLastFillerModuleAxis);
			IF stFillerModule.iq_stParameters.i_uiAxisSelected >= uiFirstFillerModuleAxis	AND
				stFillerModule.iq_stParameters.i_uiAxisSelected <= uiLastFillerModuleAxis 	AND
				stFillerModule.iq_astSubModuleAxis[uiOldAxisSelected].iq_stStatus.q_stMainAxisStatus.q_xAxisReal THEN
				IF stFillerModule.iq_stCmd.i_xOnePitchShift THEN
					stFillerModule.iq_astSubModuleAxis[uiOldAxisSelected].iq_stCmd.i_xOnePitchShift := TRUE;
					uiAutoStep	:= 150;
				ELSIF stFillerModule.iq_stCmd.i_xPhaseShift AND stFillerModule.iq_stParameters.i_rPhaseShiftDistance <> 0 THEN
					stFillerModule.iq_astSubModuleAxis[uiOldAxisSelected].iq_stParam.i_rPhaseShiftDistance 	:= stFillerModule.iq_stParameters.i_rPhaseShiftDistance;
					stFillerModule.iq_astSubModuleAxis[uiOldAxisSelected].iq_stCmd.i_xPhaseShift			:= TRUE;
					uiAutoStep	:= 180;
				END_IF
			END_IF
		ELSIF stFillerModule.iq_stStatus.q_xSynchroWithOffset AND stFillerModule.iq_stCmd.i_xPhaseCompensation THEN
			uiAutoStep	:= 300;
		END_IF

	150:(* Phase Shift Steps *)
		IF stFillerModule.iq_astSubModuleAxis[uiOldAxisSelected].iq_stStatus.q_stMainAxisStatus.q_xPhaseShiftDone THEN
			stFillerModule.iq_astSubModuleAxis[uiOldAxisSelected].iq_stCmd.i_xOnePitchShift := FALSE;
			uiAutoStep	:= 160;
		END_IF

	160:
		IF NOT stFillerModule.iq_astSubModuleAxis[uiOldAxisSelected].iq_stStatus.q_stMainAxisStatus.q_xPhaseShiftDone THEN
			uiAutoStep	:= 130;
		END_IF

	180:
		IF stFillerModule.iq_astSubModuleAxis[uiOldAxisSelected].iq_stStatus.q_stMainAxisStatus.q_xPhaseShiftDone AND NOT stFillerModule.iq_stCmd.i_xPhaseShift THEN
			stFillerModule.iq_astSubModuleAxis[uiOldAxisSelected].iq_stCmd.i_xPhaseShift 	:= FALSE;
			uiAutoStep	:= 160;
		END_IF

	300:(* Phase Offset Compensations *)
		FOR uiAxisIndex	:= uiFirstFillerModuleAxis	TO uiLastFillerModuleAxis BY 1 DO
			IF stFillerModule.iq_astSubModuleAxis[uiAxisIndex].iq_stStatus.q_stMainAxisStatus.q_xSynchroWithOffset THEN
				stFillerModule.iq_astSubModuleAxis[uiAxisIndex].iq_stCmd.i_xGear 				:= FALSE;
				stFillerModule.iq_astSubModuleAxis[uiAxisIndex].iq_stCmd.i_xPhaseCompensation	:= TRUE;
			END_IF
		END_FOR
		uiAutoStep	:= 310;

	310:
		IF NOT stFillerModule.iq_stStatus.q_xSynchroWithOffset THEN
			FOR uiAxisIndex	:= uiFirstFillerModuleAxis TO uiLastFillerModuleAxis BY 1 DO
				IF NOT stFillerModule.iq_astSubModuleAxis[uiAxisIndex].iq_stStatus.q_stMainAxisStatus.q_xVelocityControl THEN
					stFillerModule.iq_astSubModuleAxis[uiAxisIndex].iq_stCmd.i_xGear := stFillerModule.iq_astSubModuleAxis[uiAxisIndex].iq_stStatus.q_stMainAxisStatus.q_xAxisReal;
				ELSE
					stFillerModule.iq_astSubModuleAxis[uiAxisIndex].iq_stCmd.i_xGear := NOT stFillerModule.iq_stCmd.i_xVelocityAxisStop;
				END_IF
				stFillerModule.iq_astSubModuleAxis[uiAxisIndex].iq_stCmd.i_xPhaseCompensation	:= FALSE;
			END_FOR
			uiAutoStep	:= 120;
		END_IF
END_CASE

IF uiAutoStep > 120 AND EDGE(stFillerModule.iq_stCmd.i_xVelocityAxisStop) THEN
	FOR uiAxisIndex	:= uiFirstFillerModuleAxis TO uiLastFillerModuleAxis BY 1 DO
		IF stFillerModule.iq_astSubModuleAxis[uiAxisIndex].iq_stStatus.q_stMainAxisStatus.q_xVelocityControl THEN
			stFillerModule.iq_astSubModuleAxis[uiAxisIndex].iq_stCmd.i_xGear := NOT stFillerModule.iq_stCmd.i_xVelocityAxisStop;
		END_IF
	END_FOR
END_IF
END_STEP
ENTRY_ACTION
uiAutoStep	:= 0;
END_ACTION
EXIT_ACTION
stFillerModule.iq_astSubModuleAxis[CST_ModuleMasterAxis].iq_stCmd.i_xHome	:= FALSE;
stFillerModule.iq_stStatus.q_xMasterRephased :=	FALSE;
END_ACTION
TRANSITION FROM Auto TO AutoExit:=
NOT xAutoMode
END_TRANSITION
STEP AutoExit:
IF stFillerModule.iq_stStatus.q_xModuleStopped THEN
	FOR uiAxisIndex	:= uiFirstFillerModuleAxis	TO uiLastFillerModuleAxis BY 1 DO
		stFillerModule.iq_astSubModuleAxis[uiAxisIndex].iq_stCmd.i_xGear 				:= FALSE;
		stFillerModule.iq_astSubModuleAxis[uiAxisIndex].iq_stCmd.i_xPhaseCompensation	:= FALSE;
	END_FOR

	IF NOT stFillerModule.iq_stStatus.q_xRealAxesSynchronized THEN
		stFillerModule.iq_astSubModuleAxis[CST_ModuleMasterAxis].iq_stCmd.i_xGear 				:= FALSE;
		stFillerModule.iq_astSubModuleAxis[CST_ModuleMasterAxis].iq_stCmd.i_xPhaseCompensation	:= FALSE;
		xExitStep	:= NOT stFillerModule.iq_astSubModuleAxis[CST_ModuleMasterAxis].iq_stStatus.q_stMainAxisStatus.q_xSynchronized;
	END_IF
END_IF
END_STEP
TRANSITION FROM AutoExit TO ModeSelection:=
xExitStep
END_TRANSITION
(* @SFCISJUMP := 'ModeSelection' *)
STEP SubModuleCalls:
(****** TOKEN RING ALGORITHM ******)
uiTokenIndex := uiTokenIndex + 1;
IF auiAxisTokenList[uiTokenIndex] = 0 THEN
	uiTokenIndex := 0;
END_IF
uiAxisToken := auiAxisTokenList[uiTokenIndex];

(* FUBs CALLS *)
fbFillerMaster.i_xToken	:= TRUE;
fbFillerMaster;

fbMain.i_xToken			:= (uiAxisToken = CST_MainAxis OR NOT CST_AxesMultiplexingOn);	//V4.A.A.1.6.10
fbMain;

FOR uiAxisIndex := CST_FirstFillerModuleAxis TO CST_LastFillerModuleAxis DO
	IF axAxisPresent[uiAxisIndex] THEN
		CASE uiAxisIndex OF
			CST_Inlet01:
				fbInlet01.i_xToken	:= uiAxisToken = uiAxisIndex	OR NOT CST_AxesMultiplexingOn	OR stFillerModule.iq_astSubModuleAxis[uiAxisIndex].iq_stCmd.i_xCamConnected;	//V4.A.A.1.6.10
				fbInlet01.i_xParityPhasing	:= xParityPhase;
				fbInlet01;

			CST_Inlet02:
				fbInlet02.i_xToken	:= uiAxisToken = uiAxisIndex	OR NOT CST_AxesMultiplexingOn	OR stFillerModule.iq_astSubModuleAxis[uiAxisIndex].iq_stCmd.i_xCamConnected;	//V4.A.A.1.6.10
				fbInlet02.i_xParityPhasing	:= xParityPhase;
				fbInlet02;

			CST_Inlet03:
				fbInlet03.i_xToken	:= uiAxisToken = uiAxisIndex 	OR NOT CST_AxesMultiplexingOn	OR stFillerModule.iq_astSubModuleAxis[uiAxisIndex].iq_stCmd.i_xCamConnected;	//V4.A.A.1.6.10
				fbInlet03.i_xParityPhasing	:= xParityPhase;
				fbInlet03;

			CST_Inlet04:
				fbInlet04.i_xToken	:= uiAxisToken = uiAxisIndex	OR NOT CST_AxesMultiplexingOn	OR stFillerModule.iq_astSubModuleAxis[uiAxisIndex].iq_stCmd.i_xCamConnected;	//V4.A.A.1.6.10
				fbInlet04.i_xParityPhasing	:= xParityPhase;
				fbInlet04;

			CST_Inlet05:
				fbInlet05.i_xToken	:= uiAxisToken = uiAxisIndex	OR NOT CST_AxesMultiplexingOn	OR stFillerModule.iq_astSubModuleAxis[uiAxisIndex].iq_stCmd.i_xCamConnected;	//V4.A.A.1.6.10
				fbInlet05.i_xParityPhasing	:= xParityPhase;
				fbInlet05;

			CST_Inlet06:
				fbInlet06.i_xToken	:= uiAxisToken = uiAxisIndex	OR NOT CST_AxesMultiplexingOn	OR stFillerModule.iq_astSubModuleAxis[uiAxisIndex].iq_stCmd.i_xCamConnected;	//V4.A.A.1.6.10
				fbInlet06.i_xParityPhasing	:= xParityPhase;
				fbInlet06;

			CST_Inlet07:
				fbInlet07.i_xToken	:= uiAxisToken = uiAxisIndex	OR NOT CST_AxesMultiplexingOn	OR stFillerModule.iq_astSubModuleAxis[uiAxisIndex].iq_stCmd.i_xCamConnected;	//V4.A.A.1.6.10
				fbInlet07.i_xParityPhasing	:= xParityPhase;
				fbInlet07;

			CST_Inlet08:
				fbInlet08.i_xToken	:= uiAxisToken = uiAxisIndex	OR NOT CST_AxesMultiplexingOn	OR stFillerModule.iq_astSubModuleAxis[uiAxisIndex].iq_stCmd.i_xCamConnected;	//V4.A.A.1.6.10
				fbInlet08.i_xParityPhasing	:= xParityPhase;
				fbInlet08;

			CST_Inlet09:
				fbInlet09.i_xToken	:= uiAxisToken = uiAxisIndex	OR NOT CST_AxesMultiplexingOn	OR stFillerModule.iq_astSubModuleAxis[uiAxisIndex].iq_stCmd.i_xCamConnected;	//V4.A.A.1.6.10
				fbInlet09.i_xParityPhasing	:= xParityPhase;
				fbInlet09;

			CST_Inlet10:
				fbInlet10.i_xToken	:= uiAxisToken = uiAxisIndex	OR NOT CST_AxesMultiplexingOn	OR stFillerModule.iq_astSubModuleAxis[uiAxisIndex].iq_stCmd.i_xCamConnected;	//V4.A.A.1.6.10
				fbInlet10.i_xParityPhasing	:= xParityPhase;
				fbInlet10;

			CST_Outlet01:
				fbOutlet01.i_xToken	:= uiAxisToken = uiAxisIndex	OR NOT CST_AxesMultiplexingOn	OR stFillerModule.iq_astSubModuleAxis[uiAxisIndex].iq_stCmd.i_xCamConnected;	//V4.A.A.1.6.10
				fbOutlet01.i_xParityPhasing	:= xParityPhase;
				fbOutlet01;

			CST_Outlet02:
				fbOutlet02.i_xToken	:= uiAxisToken = uiAxisIndex	OR NOT CST_AxesMultiplexingOn	OR stFillerModule.iq_astSubModuleAxis[uiAxisIndex].iq_stCmd.i_xCamConnected;	//V4.A.A.1.6.10
				fbOutlet02.i_xParityPhasing	:= xParityPhase;
				fbOutlet02;

			CST_Outlet03:
				fbOutlet03.i_xToken	:= uiAxisToken = uiAxisIndex	OR NOT CST_AxesMultiplexingOn	OR stFillerModule.iq_astSubModuleAxis[uiAxisIndex].iq_stCmd.i_xCamConnected;	//V4.A.A.1.6.10
				fbOutlet03.i_xParityPhasing	:= xParityPhase;
				fbOutlet03;

			CST_Outlet04:
				fbOutlet04.i_xToken	:= uiAxisToken = uiAxisIndex	OR NOT CST_AxesMultiplexingOn	OR stFillerModule.iq_astSubModuleAxis[uiAxisIndex].iq_stCmd.i_xCamConnected;	//V4.A.A.1.6.10
				fbOutlet04.i_xParityPhasing	:= xParityPhase;
				fbOutlet04;

			CST_Outlet05:
				fbOutlet05.i_xToken	:= uiAxisToken = uiAxisIndex	OR NOT CST_AxesMultiplexingOn	OR stFillerModule.iq_astSubModuleAxis[uiAxisIndex].iq_stCmd.i_xCamConnected;	//V4.A.A.1.6.10
				fbOutlet05.i_xParityPhasing	:= xParityPhase;
				fbOutlet05;

			CST_Outlet06:
				fbOutlet06.i_xToken	:= uiAxisToken = uiAxisIndex	OR NOT CST_AxesMultiplexingOn	OR stFillerModule.iq_astSubModuleAxis[uiAxisIndex].iq_stCmd.i_xCamConnected;	//V4.A.A.1.6.10
				fbOutlet06.i_xParityPhasing	:= xParityPhase;
				fbOutlet06;
		END_CASE
	END_IF
END_FOR
END_STEP
STEP SetException:
(* Set Exception Action *)
fbMpAlarmXCore(MpLink := ADR(gFillerAlarmXCoreLink), Enable := TRUE);
stFillerModule.iq_stStatus.q_xAlarmXCoreEnabled	:= fbMpAlarmXCore.Active;

(* Axis errors *)
fbMasterError(i_xConditions	:= stFillerModule.iq_astSubModuleAxis[CST_ModuleMasterAxis].iq_stStatus.q_stMainAxisStatus.q_xError);

fbMainAxisError(i_xConditions		:= stFillerModule.iq_astSubModuleAxis[CST_MainAxis].iq_stStatus.q_stMainAxisStatus.q_xError);
fbMainAxisLagError(i_xConditions	:= stFillerModule.iq_astSubModuleAxis[CST_MainAxis].iq_stStatus.q_stMainAxisStatus.q_xLagError);

IF axAxisPresent[CST_Inlet01] THEN
	fbInlet01Error(i_xConditions	:= stFillerModule.iq_astSubModuleAxis[CST_Inlet01].iq_stStatus.q_stMainAxisStatus.q_xError);
	fbInlet01LagError(i_xConditions	:= stFillerModule.iq_astSubModuleAxis[CST_Inlet01].iq_stStatus.q_stMainAxisStatus.q_xLagError);
END_IF

IF axAxisPresent[CST_Inlet02] THEN
	fbInlet02Error(i_xConditions	:= stFillerModule.iq_astSubModuleAxis[CST_Inlet02].iq_stStatus.q_stMainAxisStatus.q_xError);
	fbInlet02LagError(i_xConditions	:= stFillerModule.iq_astSubModuleAxis[CST_Inlet02].iq_stStatus.q_stMainAxisStatus.q_xLagError);
END_IF

IF axAxisPresent[CST_Inlet03] THEN
	fbInlet03Error(i_xConditions	:= stFillerModule.iq_astSubModuleAxis[CST_Inlet03].iq_stStatus.q_stMainAxisStatus.q_xError);
	fbInlet03LagError(i_xConditions	:= stFillerModule.iq_astSubModuleAxis[CST_Inlet03].iq_stStatus.q_stMainAxisStatus.q_xLagError);
END_IF

IF axAxisPresent[CST_Inlet04] THEN
	fbInlet04Error(i_xConditions	:= stFillerModule.iq_astSubModuleAxis[CST_Inlet04].iq_stStatus.q_stMainAxisStatus.q_xError);
	fbInlet04LagError(i_xConditions	:= stFillerModule.iq_astSubModuleAxis[CST_Inlet04].iq_stStatus.q_stMainAxisStatus.q_xLagError);
END_IF

IF axAxisPresent[CST_Inlet05] THEN
	fbInlet05Error(i_xConditions	:= stFillerModule.iq_astSubModuleAxis[CST_Inlet05].iq_stStatus.q_stMainAxisStatus.q_xError);
	fbInlet05LagError(i_xConditions	:= stFillerModule.iq_astSubModuleAxis[CST_Inlet05].iq_stStatus.q_stMainAxisStatus.q_xLagError);
END_IF

IF axAxisPresent[CST_Inlet06] THEN
	fbInlet06Error(i_xConditions	:= stFillerModule.iq_astSubModuleAxis[CST_Inlet06].iq_stStatus.q_stMainAxisStatus.q_xError);
	fbInlet06LagError(i_xConditions	:= stFillerModule.iq_astSubModuleAxis[CST_Inlet06].iq_stStatus.q_stMainAxisStatus.q_xLagError);
END_IF

IF axAxisPresent[CST_Inlet07] THEN
	fbInlet07Error(i_xConditions	:= stFillerModule.iq_astSubModuleAxis[CST_Inlet07].iq_stStatus.q_stMainAxisStatus.q_xError);
	fbInlet07LagError(i_xConditions	:= stFillerModule.iq_astSubModuleAxis[CST_Inlet07].iq_stStatus.q_stMainAxisStatus.q_xLagError);
END_IF

IF axAxisPresent[CST_Inlet08] THEN
	fbInlet08Error(i_xConditions	:= stFillerModule.iq_astSubModuleAxis[CST_Inlet08].iq_stStatus.q_stMainAxisStatus.q_xError);
	fbInlet08LagError(i_xConditions	:= stFillerModule.iq_astSubModuleAxis[CST_Inlet08].iq_stStatus.q_stMainAxisStatus.q_xLagError);
END_IF

IF axAxisPresent[CST_Inlet09] THEN
	fbInlet09Error(i_xConditions	:= stFillerModule.iq_astSubModuleAxis[CST_Inlet09].iq_stStatus.q_stMainAxisStatus.q_xError);
	fbInlet09LagError(i_xConditions	:= stFillerModule.iq_astSubModuleAxis[CST_Inlet09].iq_stStatus.q_stMainAxisStatus.q_xLagError);
END_IF

IF axAxisPresent[CST_Inlet10] THEN
	fbInlet10Error(i_xConditions	:= stFillerModule.iq_astSubModuleAxis[CST_Inlet10].iq_stStatus.q_stMainAxisStatus.q_xError);
	fbInlet10LagError(i_xConditions	:= stFillerModule.iq_astSubModuleAxis[CST_Inlet10].iq_stStatus.q_stMainAxisStatus.q_xLagError);
END_IF

IF axAxisPresent[CST_Outlet01] THEN
	fbOutlet01Error(i_xConditions		:= stFillerModule.iq_astSubModuleAxis[CST_Outlet01].iq_stStatus.q_stMainAxisStatus.q_xError);
	fbOutlet01LagError(i_xConditions	:= stFillerModule.iq_astSubModuleAxis[CST_Outlet01].iq_stStatus.q_stMainAxisStatus.q_xLagError);
END_IF

IF axAxisPresent[CST_Outlet02] THEN
	fbOutlet02Error(i_xConditions		:= stFillerModule.iq_astSubModuleAxis[CST_Outlet02].iq_stStatus.q_stMainAxisStatus.q_xError);
	fbOutlet02LagError(i_xConditions	:= stFillerModule.iq_astSubModuleAxis[CST_Outlet02].iq_stStatus.q_stMainAxisStatus.q_xLagError);
END_IF

IF axAxisPresent[CST_Outlet03] THEN
	fbOutlet03Error(i_xConditions		:= stFillerModule.iq_astSubModuleAxis[CST_Outlet03].iq_stStatus.q_stMainAxisStatus.q_xError);
	fbOutlet03LagError(i_xConditions	:= stFillerModule.iq_astSubModuleAxis[CST_Outlet03].iq_stStatus.q_stMainAxisStatus.q_xLagError);
END_IF

IF axAxisPresent[CST_Outlet04] THEN
	fbOutlet04Error(i_xConditions		:= stFillerModule.iq_astSubModuleAxis[CST_Outlet04].iq_stStatus.q_stMainAxisStatus.q_xError);
	fbOutlet04LagError(i_xConditions	:= stFillerModule.iq_astSubModuleAxis[CST_Outlet04].iq_stStatus.q_stMainAxisStatus.q_xLagError);
END_IF

IF axAxisPresent[CST_Outlet05] THEN
	fbOutlet05Error(i_xConditions		:= stFillerModule.iq_astSubModuleAxis[CST_Outlet05].iq_stStatus.q_stMainAxisStatus.q_xError);
	fbOutlet05LagError(i_xConditions	:= stFillerModule.iq_astSubModuleAxis[CST_Outlet05].iq_stStatus.q_stMainAxisStatus.q_xLagError);
END_IF

IF axAxisPresent[CST_Outlet06] THEN
	fbOutlet06Error(i_xConditions		:= stFillerModule.iq_astSubModuleAxis[CST_Outlet06].iq_stStatus.q_stMainAxisStatus.q_xError);
	fbOutlet06LagError(i_xConditions	:= stFillerModule.iq_astSubModuleAxis[CST_Outlet06].iq_stStatus.q_stMainAxisStatus.q_xLagError);
END_IF

fbEmergencyStopAlarm(i_xConditions	:= NOT stFillerModule.iq_stCmd.i_xEnable);
fbQuickStopFromPlc(i_xConditions	:= NOT stFillerModule.iq_stCmd.i_xExternalQuickStop);
END_STEP
STEP Output:
(* Modalities Bits *)
stFillerModule.iq_stStatus.q_xNoOpActive			:= xNoOpActive;
stFillerModule.iq_stStatus.q_xAutoActive 			:= xAutoActive;
stFillerModule.iq_stStatus.q_xPositioningActive 	:= xPositioningActive;
stFillerModule.iq_stStatus.q_xSelHomingActive 		:= xSelHomingActive;
stFillerModule.iq_stStatus.q_xBrakeReleaseActive 	:= xBrakeReleaseActive;
stFillerModule.iq_stStatus.q_xSlowMotionActive 		:= xSlowMotionActive;
stFillerModule.iq_stStatus.q_xJogMultiActive 		:= xJogMultiActive;
stFillerModule.iq_stStatus.q_xAutoMultiActive 		:= xAutoMultiActive;
stFillerModule.iq_stStatus.q_xStepByStepActive 		:= xStepByStepActive;
stFillerModule.iq_stStatus.q_xVelocityActive 		:= xVelocityActive;
stFillerModule.iq_stStatus.q_xThirdPartySetupActive	:= xThirdPartySetupActive;
stFillerModule.iq_stStatus.q_xInductionSetupActive	:= xInductionSetupActive;

stFillerModule.iq_stStatus.q_xModuleStartFbk	:= (xAutoMultiActive	AND stFillerModule.iq_stCmd.i_xStart)	OR
													(xJogMultiActive	AND stFillerModule.iq_stCmd.i_xJogPB)	OR
													(xSlowMotionActive	AND stFillerModule.iq_stCmd.i_xJogPB);

CASE uiSlowAxisIndex OF
	CST_ModuleMasterAxis:
		stFillerModule.iq_stStatus.q_xModulePowered				:= xModulePowered;
		stFillerModule.iq_stStatus.q_xRealAxesReadyForACommand	:= xRealAxesReadyForACommand;
		stFillerModule.iq_stStatus.q_xSynchroWithOffset			:= xSynchroWithOffset;
		stFillerModule.iq_stStatus.q_xModuleStopped				:= xModuleStopped;
		stFillerModule.iq_stStatus.q_xRealAxesSynchronized		:= xRealAxesSynchronized;
		stFillerModule.iq_stStatus.q_xPhaseShiftDone			:= xPhaseShiftDone;
		stFillerModule.iq_stStatus.q_xSelHomingDone				:= xSelHomingDone;
		stFillerModule.iq_stStatus.q_xModuleHomed				:= xModuleHomed;
		stFillerModule.iq_stStatus.q_xInitDone					:= xModuleInitialized;

		// Module Velocity
		stFillerModule.iq_stStatus.q_rVelocity					:= rModuleVelocity;
		rModuleVelocity											:= ABS(stFillerModule.iq_astSubModuleAxis[uiSlowAxisIndex].iq_stStatus.q_stMainAxisStatus.q_rVelocity);
		usiMasterStatus											:= usiMasterTempStatus;
		usiMasterTempStatus										:= usiMasterRequest;

	CST_FirstFillerModuleAxis..CST_LastFillerModuleAxis:
		IF NOT stFillerModule.iq_astSubModuleAxis[uiSlowAxisIndex].iq_stStatus.q_stMainAxisStatus.q_xPowerSupply	AND
			stFillerModule.iq_astSubModuleAxis[uiSlowAxisIndex].iq_stStatus.q_stMainAxisStatus.q_xAxisReal			THEN

			IF NOT stFillerModule.iq_astSubModuleAxis[uiSlowAxisIndex].iq_stStatus.q_stMainAxisStatus.q_xVelocityControl THEN
				rModuleVelocity	:= MAX(rModuleVelocity, ABS(stFillerModule.iq_astSubModuleAxis[uiSlowAxisIndex].iq_stStatus.q_stMainAxisStatus.q_rVelocity));
			END_IF

			// Master management
			IF	usiMasterRequest = LOCAL_MASTER THEN
				IF stFillerModule.iq_astSubModuleAxis[uiSlowAxisIndex].iq_stStatus.q_stMainAxisStatus.q_udiMasterAxisLink <> ADR(gFillerModuleMasterLink) AND usiMasterTempStatus <> UNKNOWN THEN
					usiMasterTempStatus := UNKNOWN;
				END_IF
			ELSIF usiMasterRequest = GLOBAL_MASTER THEN
				IF stFillerModule.iq_astSubModuleAxis[uiSlowAxisIndex].iq_stStatus.q_stMainAxisStatus.q_udiMasterAxisLink <> ADR(gMasterLink) AND usiMasterTempStatus <> UNKNOWN THEN
					usiMasterTempStatus := UNKNOWN;
				END_IF
			ELSE
				usiMasterStatus	:= UNKNOWN;
			END_IF

			// Module Initialized Memory
			xModuleInitialized	:= xModuleInitialized AND
									stFillerModule.iq_astSubModuleAxis[uiSlowAxisIndex].iq_stStatus.q_stMainAxisStatus.q_xInitDone;

			// Axis Homed cumulative memory
			xModuleHomed		:= xModuleHomed AND
									stFillerModule.iq_astSubModuleAxis[uiSlowAxisIndex].iq_stStatus.q_stMainAxisStatus.q_xIsHomed;

			// Axis stopped cumulative memory
			xModuleStopped		:= xModuleStopped AND
									(stFillerModule.iq_astSubModuleAxis[uiSlowAxisIndex].iq_stStatus.q_stMainAxisStatus.q_xStopped OR NOT
									stFillerModule.iq_astSubModuleAxis[uiSlowAxisIndex].iq_stStatus.q_stMainAxisStatus.q_xPoweredOn);

			// Ready for a command cumulative memory
			xRealAxesReadyForACommand	:= xRealAxesReadyForACommand AND stFillerModule.iq_astSubModuleAxis[uiSlowAxisIndex].iq_stStatus.q_stMainAxisStatus.q_xReadyForACommand;

			IF NOT stFillerModule.iq_astSubModuleAxis[uiSlowAxisIndex].iq_stStatus.q_stMainAxisStatus.q_xAxisDisabled THEN
				// Axis syncrhonized cumulative memory
				xRealAxesSynchronized	:= xRealAxesSynchronized	AND stFillerModule.iq_astSubModuleAxis[uiSlowAxisIndex].iq_stStatus.q_stMainAxisStatus.q_xSynchronized;
				// There is at least One Axis with a phase offset pending
				xSynchroWithOffset		:= xSynchroWithOffset		OR stFillerModule.iq_astSubModuleAxis[uiSlowAxisIndex].iq_stStatus.q_stMainAxisStatus.q_xSynchroWithOffset;
				// Phase shift done
				xPhaseShiftDone			:= xPhaseShiftDone 	OR (stFillerModule.iq_astSubModuleAxis[uiSlowAxisIndex].iq_stStatus.q_stMainAxisStatus.q_xPhaseShiftDone AND stFillerModule.iq_astSubModuleAxis[uiSlowAxisIndex].iq_stCmd.i_xPhaseShift);
			END_IF
		END_IF
	ELSE
		xRealAxesReadyForACommand	:= TRUE;
		xSynchroWithOffset			:= FALSE;
		xModuleStopped				:= TRUE;
		xRealAxesSynchronized		:= TRUE;
		xPhaseShiftDone				:= FALSE;
		xSelHomingDone				:= FALSE;
		xModuleHomed				:= TRUE;
		xModuleInitialized			:= TRUE;
END_CASE

stFillerModule.iq_stStatus.q_xModulePowered		:= FALSE;
stFillerModule.iq_stStatus.q_xReactionActive	:= xReactionActive;

FOR uiAxisIndex := uiFirstFillerModuleAxis TO uiLastFillerModuleAxis BY 1 DO
	// Axis powered cumulative memory
	stFillerModule.iq_stStatus.q_xModulePowered	:= stFillerModule.iq_stStatus.q_xModulePowered		OR
													(stFillerModule.iq_astSubModuleAxis[uiAxisIndex].iq_stStatus.q_stMainAxisStatus.q_xPoweredOn 		AND
													NOT stFillerModule.iq_astSubModuleAxis[uiAxisIndex].iq_stStatus.q_stMainAxisStatus.q_xPowerSupply 	AND
							 						stFillerModule.iq_astSubModuleAxis[uiAxisIndex].iq_stStatus.q_stMainAxisStatus.q_xAxisReal);
END_FOR

stFillerModule.iq_stStatus.q_xModuleSynchronized		:= stFillerModule.iq_stStatus.q_xRealAxesSynchronized;

(********* Wheel position calculation **********)
fbFillerAbsPos( (*//V4.A.A.1.6.12e*)
i_xEnable					:= CFG_MC.Mechanical.ReferenceId.Filler <> 0, (*//V4.A.A.1.6.12e*)
i_pstAxis					:= stFillerModule.iq_astSubModuleAxis[CFG_MC.Mechanical.ReferenceId.Filler], (*//V4.A.A.1.6.12e*)
i_xPositionSensor			:= stFillerModule.iq_stCmd.i_xFillerAbsolutePositionSensor, (*//V4.A.A.1.6.12e*)//V1.7.2
i_uiAbsolutePositionOffset	:= stFillerModule.iq_stParameters.i_uiFillerAbsolutePositionOffset, (*//V4.A.A.1.6.12e*)
i_uiStepsNumber				:= stFillerModule.iq_stParameters.i_uiFillerStepsNumber (*//V4.A.A.1.6.12e*)
); (*//V4.A.A.1.6.12e*)

(********* Rinser position calculation **********)//V4.A.A.1.7.0 Foot
fbRinserAbsPos( //V4.A.A.1.7.0 Foot
i_xEnable					:= CFG_MC.Mechanical.ReferenceId.Rinser <> 0, //V4.A.A.1.7.0 Foot
i_pstAxis					:= stFillerModule.iq_astSubModuleAxis[CFG_MC.Mechanical.ReferenceId.Rinser], //V4.A.A.1.7.0 Foot
i_xPositionSensor			:= stFillerModule.iq_stCmd.i_xRinserFillerAbsolutePosSensor AND EDGEPOS(MC_InputOutput.Network.Machine.Status.MachineClockA) AND MC_InputOutput.Network.Machine.Status.MachineRunning,//V4.A.A.1.7.0 Foot
i_uiAbsolutePositionOffset	:= stFillerModule.iq_stParameters.i_uiRinserAbsolutePositionOffset,//V4.A.A.1.7.0 Foot
i_uiStepsNumber				:= stFillerModule.iq_stParameters.i_uiRinserStepsNumber //V4.A.A.1.7.0 Foot
);
(********* Doser position calculation **********)//V4.A.A.1.7.0 Foot
fbDoserAbsPos( //V4.A.A.1.7.0 Foot
i_xEnable					:= CFG_MC.Mechanical.ReferenceId.Doser <> 0, //V4.A.A.1.7.0 Foot
i_pstAxis					:= stFillerModule.iq_astSubModuleAxis[CFG_MC.Mechanical.ReferenceId.Doser], //V4.A.A.1.7.0 Foot
i_xPositionSensor			:= stFillerModule.iq_stCmd.i_xDoserAbsolutePositionSensor AND EDGEPOS(MC_InputOutput.Network.Machine.Status.MachineClockA) AND MC_InputOutput.Network.Machine.Status.MachineRunning,//V4.A.A.1.7.0 Foot
i_uiAbsolutePositionOffset	:= stFillerModule.iq_stParameters.i_uiDoserPositionOffset,//V4.A.A.1.7.0 Foot
i_uiStepsNumber				:= stFillerModule.iq_stParameters.i_uiDoserStepsNumber //V4.A.A.1.7.0 Foot
);
(********* Capper position calculation **********)
fbCapperAbsPos( //V4.A.A.1.6.12e
i_xEnable					:= CFG_MC.Mechanical.ReferenceId.Capper <> 0, (*//V4.A.A.1.6.12e*)
i_pstAxis					:= stFillerModule.iq_astSubModuleAxis[CFG_MC.Mechanical.ReferenceId.Capper], (*//V4.A.A.1.6.12e*)
i_xPositionSensor			:= stFillerModule.iq_stCmd.i_xCapperAbsolutePositionSensor AND EDGEPOS(MC_InputOutput.Network.Machine.Status.MachineClockA) AND MC_InputOutput.Network.Machine.Status.MachineRunning, (*//V4.A.A.1.6.12e*)
i_uiAbsolutePositionOffset	:= stFillerModule.iq_stParameters.i_uiCapperAbsolutePositionOffset, (*//V4.A.A.1.6.12e*)
i_uiStepsNumber				:= stFillerModule.iq_stParameters.i_uiCapperStepsNumber (*//V4.A.A.1.6.12e*)
);
(********* Crowner position calculation **********)//V4.A.A.1.7.0 Foot
fbCrownerAbsPos( //V4.A.A.1.7.0 Foot
i_xEnable					:= CFG_MC.Mechanical.ReferenceId.Crowner <> 0, //V4.A.A.1.7.0 Foot
i_pstAxis					:= stFillerModule.iq_astSubModuleAxis[CFG_MC.Mechanical.ReferenceId.Crowner],//V4.A.A.1.7.0 Foot
i_xPositionSensor			:= stFillerModule.iq_stCmd.i_xCrownerAbsolutePositionSensor AND EDGEPOS(MC_InputOutput.Network.Machine.Status.MachineClockA) AND MC_InputOutput.Network.Machine.Status.MachineRunning,//V4.A.A.1.7.0 Foot
i_uiAbsolutePositionOffset	:= stFillerModule.iq_stParameters.i_uiCrownerAbsolutePosOffset,//V4.A.A.1.7.0 Foot
i_uiStepsNumber				:= stFillerModule.iq_stParameters.i_uiCrownerStepsNumber //V4.A.A.1.7.0 Foot
);

IF EDGEPOS(stFillerModule.iq_astSubModuleAxis[CST_MainAxis].iq_stCmd.i_xGear) THEN
	lrTempOldPosition := stFillerModule.iq_astSubModuleAxis[CST_MainAxis].iq_stStatus.q_stMainAxisStatus.q_lrPosition;
END_IF

IF stFillerModule.iq_astSubModuleAxis[CST_MainAxis].iq_stCmd.i_xGear AND NOT stFillerModule.iq_astSubModuleAxis[CST_MainAxis].iq_stStatus.q_stMainAxisStatus.q_xSynchronized THEN
	lrTempPosDiff := lrTempOldPosition - stFillerModule.iq_astSubModuleAxis[CST_ModuleMasterAxis].iq_stStatus.q_stMainAxisStatus.q_lrPosition;

	IF (lrTempPosDiff > 0	AND lrTempPosDiff < 3.0) OR
		(lrTempPosDiff < 0	AND lrTempPosDiff + 360.0 < 3.0) THEN
		iTempParity := TRUNC((lrFillerAbsolutePosition + lrTempPosDiff) / 360.0); (*//V4.A.A.1.6.12e*)
	ELSE
		iTempParity := TRUNC((lrFillerAbsolutePosition + FC_LongRealReminder(stFillerModule.iq_astSubModuleAxis[CST_ModuleMasterAxis].iq_stStatus.q_stMainAxisStatus.q_lrPosition - lrTempOldPosition, 360.0, 0.0)) / 360.0); (*//V4.A.A.1.6.12e*)
	END_IF
ELSE
	iTempParity := TRUNC(lrFillerAbsolutePosition / 360.0); (*//V4.A.A.1.6.12e*)
END_IF

xParityPhase := NOT iTempParity.0;
//xParityPhase		:= FC_Parity(IN_Value := INT_TO_DINT(TRUNC(lrAbsolutePosition / 360.0)));

(* Position valid condition *)
stFillerModule.iq_stStatus.q_xFillerAbsolutePositionValid	:= fbFillerAbsPos.q_xPositionValid; (*//V4.A.A.1.6.12e*)

IF fbFillerAbsPos.q_xPositionValid THEN (*//V4.A.A.1.6.12e*)
	stFillerModule.iq_stStatus.q_lrFillerAbsolutePosition	:= fbFillerAbsPos.q_lrAbsolutePosition; (*//V4.A.A.1.6.12e*)
ELSE
	stFillerModule.iq_stStatus.q_lrFillerAbsolutePosition	:= 0; (*//V4.A.A.1.6.12e*)
END_IF
//V4.A.A.1.7.0 Foot
stFillerModule.iq_stStatus.q_xRinserAbsolutePositionValid	:= fbRinserAbsPos.q_xPositionValid;//V4.A.A.1.7.0 Foot

IF fbRinserAbsPos.q_xPositionValid THEN//V4.A.A.1.7.0 Foot
	stFillerModule.iq_stStatus.q_lrRinserAbsolutePosition	:= fbRinserAbsPos.q_lrAbsolutePosition;//V4.A.A.1.7.0 Foot
ELSE
	stFillerModule.iq_stStatus.q_lrRinserAbsolutePosition	:= 0;//V4.A.A.1.7.0 Foot
END_IF
//V4.A.A.1.7.0 Foot
stFillerModule.iq_stStatus.q_xDoserAbsolutePositionValid	:= fbDoserAbsPos.q_xPositionValid;//V4.A.A.1.7.0 Foot

IF fbDoserAbsPos.q_xPositionValid THEN//V4.A.A.1.7.0 Foot
	stFillerModule.iq_stStatus.q_lrDoserAbsolutePosition	:= fbDoserAbsPos.q_lrAbsolutePosition;//V4.A.A.1.7.0 Foot
ELSE
	stFillerModule.iq_stStatus.q_lrDoserAbsolutePosition	:= 0;//V4.A.A.1.7.0 Foot
END_IF
//V4.A.A.1.7.0 Foot
stFillerModule.iq_stStatus.q_xCapperAbsolutePositionValid	:= fbCapperAbsPos.q_xPositionValid; (*//V4.A.A.1.6.12e*)

IF fbCapperAbsPos.q_xPositionValid THEN (*//V4.A.A.1.6.12e*)
	stFillerModule.iq_stStatus.q_lrCapperAbsolutePosition	:= fbCapperAbsPos.q_lrAbsolutePosition; (*//V4.A.A.1.6.12e*)
ELSE
	stFillerModule.iq_stStatus.q_lrCapperAbsolutePosition	:= 0; (*//V4.A.A.1.6.12e*)
END_IF
//V4.A.A.1.7.0 Foot
stFillerModule.iq_stStatus.q_xCrownerAbsolutePositionValid	:= fbCrownerAbsPos.q_xPositionValid;//V4.A.A.1.7.0 Foot

IF fbCrownerAbsPos.q_xPositionValid THEN//V4.A.A.1.7.0 Foot
	stFillerModule.iq_stStatus.q_lrCrownerAbsolutePosition	:= fbCrownerAbsPos.q_lrAbsolutePosition;//V4.A.A.1.7.0 Foot
ELSE
	stFillerModule.iq_stStatus.q_lrCrownerAbsolutePosition	:= 0;//V4.A.A.1.7.0 Foot
END_IF
END_STEP
TRANSITION FROM (Input,SubModuleCalls,SetException,Output) TO Disabled:=
FALSE
END_TRANSITION
STEP Disabled:
stFillerModule.iq_stStatus.q_xAlarmXCoreEnabled	:= TRUE;
END_STEP
TRANSITION FROM Disabled TO Init:=
FALSE
END_TRANSITION
(* @SFCISJUMP := 'Init' *)
END_PROGRAM
```

#### Init.st
```iecst
PROGRAM _INIT
	stFillerModule	ACCESS ADR(VAR_Machine.stFillerModule);
END_PROGRAM
```

### Program Logical/30_MC/Task/Cyclic02/MC_INLET (IEC) - MC_INLET - C#1 0.8ms or C#2 10.4ms

#### Variables.var
```iecst
(* Input Variables *)
VAR
	xInputAuto : BOOL;
	xInputVelocity : BOOL;
	xInputJogMulti : BOOL;
	xInputAutoMulti : BOOL;
	xInputSelHoming : BOOL;
	xInputThirdPartySetup : BOOL;
	xInputInductionSetup : BOOL;
	xInputPositioning : BOOL;
	xInputSlowMotion : BOOL;
	xInputBrakeRelease : BOOL;
	xInputStepByStep : BOOL;
END_VAR
(*Modality Bits*)
VAR
	xModeReady : BOOL;
	xExitStep : BOOL; (*Exit Step Variables*)
	xAutoMode : BOOL; (*Auto Mode Command Variables*)
	xVelocityMode : BOOL;
	xPositioningMode : BOOL; (*Positioning Mode Command Variable*)
	xThirdPartySetupMode : BOOL;
	xInductionSetupMode : BOOL;
	xSelectiveHomingMode : BOOL; (*Selective Homing Command Variable*)
	xBrakeReleaseMode : BOOL;
	xAutoMultiMode : BOOL;
	xJogMultiMode : BOOL;
	xStepByStepMode : BOOL;
	xSlowMotionMode : BOOL;
	xModulePowered : BOOL;
	xRealAxesReadyForACommand : BOOL;
	xSynchroWithOffset : BOOL;
	xModuleStopped : BOOL;
	xRealAxesSynchronized : BOOL;
	xPhaseShiftDone : BOOL;
	xSelHomingDone : BOOL;
	xModuleInitialized : BOOL;
	xModuleHomed : BOOL;
END_VAR
(*Active Modality Bits*)
VAR
	xNoOpActive : BOOL;
	xAutoActive : BOOL;
	xPositioningActive : BOOL;
	xThirdPartySetupActive : BOOL;
	xInductionSetupActive : BOOL;
	xSelHomingActive : BOOL;
	xBrakeReleaseActive : BOOL;
	xVelocityActive : BOOL;
	xSlowMotionActive : BOOL;
	xJogMultiActive : BOOL;
	xAutoMultiActive : BOOL;
	xStepByStepActive : BOOL;
END_VAR
(*Axes presence*)
VAR
	axAxisPresent : ARRAY[CST_FirstInletModuleAxis..CST_LastInletModuleAxis] OF BOOL := [9(FALSE)];
END_VAR
(*Local master management*)
VAR
	usiMasterRequest : E_MasterStatus;
	usiMasterStatus : E_MasterStatus;
	usiMasterTempStatus : E_MasterStatus;
END_VAR
(*FB axis Declarations*)
VAR
	fbInletMaster : FB_GeneralAxis;
	fbMain : FB_GeneralAxis;
	fbInlet01 : FB_GeneralAxis;
	fbInlet02 : FB_GeneralAxis;
	fbInlet03 : FB_GeneralAxis;
	fbInlet04 : FB_GeneralAxis;
	fbOutlet01 : FB_GeneralAxis;
	fbOutlet02 : FB_GeneralAxis;
	fbOutlet03 : FB_GeneralAxis;
	fbOutlet04 : FB_GeneralAxis;
END_VAR
(*Local Module Struct*)
VAR
	stInletModule : REFERENCE TO ST_InletModuleInterface; (*Inlet Module Interface Variables*)
	fbMpAlarmXCore : MpAlarmXCore;
END_VAR
(*Alarms bits*)
VAR
	fbQuickStopFromPlc : FB_ExceptionAlarmX;
	fbMasterError : FB_ExceptionAlarmX;
	fbMainAxisLagError : FB_ExceptionAlarmX;
	fbMainAxisError : FB_ExceptionAlarmX;
	fbInlet01LagError : FB_ExceptionAlarmX;
	fbInlet02LagError : FB_ExceptionAlarmX;
	fbInlet03LagError : FB_ExceptionAlarmX;
	fbInlet04LagError : FB_ExceptionAlarmX;
	fbOutlet01LagError : FB_ExceptionAlarmX;
	fbOutlet02LagError : FB_ExceptionAlarmX;
	fbOutlet03LagError : FB_ExceptionAlarmX;
	fbOutlet04LagError : FB_ExceptionAlarmX;
	fbInlet01Error : FB_ExceptionAlarmX;
	fbInlet02Error : FB_ExceptionAlarmX;
	fbInlet03Error : FB_ExceptionAlarmX;
	fbInlet04Error : FB_ExceptionAlarmX;
	fbOutlet01Error : FB_ExceptionAlarmX;
	fbOutlet02Error : FB_ExceptionAlarmX;
	fbOutlet03Error : FB_ExceptionAlarmX;
	fbOutlet04Error : FB_ExceptionAlarmX;
	fbEmergencyStopAlarm : FB_ExceptionAlarmX;
END_VAR
(*Local Variables*)
VAR
	xPositionValid : BOOL;
	xReactionActive : BOOL;
	uiAxisIndex : UINT; (*Axis Index*)
	uiOldAxisSelected : UINT;
	uiNextHomingPositionIndex : UINT; (*Temp var for initializing homing position chain*)
	uiFirstInletModuleAxis : UINT; (*First present axis index in Inlet module*)
	uiLastInletModuleAxis : UINT; (*Last present axis index in Inlet module*)
	uiNumberOfSteps : UINT;
	uiAxisToken : UINT;
	uiSlowAxisIndex : UINT;
	rModuleVelocity : REAL;
	rAxisDistance : REAL;
	lrAbsolutePosition : LREAL;
	lrIncrement : LREAL;
	lrOldPosition : LREAL;
	tonPositDone : TON;
	tofReactionActive : TOF;
	axPresentIndex : USINT;
END_VAR
(*Sequencer Steps*)
VAR
	uiVelocityStep : UINT;
	uiAutoStep : UINT;
	uiPositioningStep : UINT;
	uiInductionSetupStep : UINT;
	uiThirdPartySetupStep : UINT;
	uiSelectiveHomeStep : UINT;
	uiBrakeReleaseStep : UINT;
	uiSlowMotionStep : UINT;
	uiJogMulti : UINT;
	uiAutoMulti : UINT;
	uiStepByStep : UINT;
	auiAxisTokenList : ARRAY[0..20] OF UINT;
	uiTokenIndex : UINT;
END_VAR
```
